// TIA Portal V15.1 export
// export: Created 2024-05-17T05:38:21.716242Z, ExportSetting WithDefaults, DisplayName Totally Integrated Automation Portal, DisplayVersion V15.1 Update 5, DisplayName TIA Portal Openness, DisplayVersion V15.1 Update 5, DisplayName SINAMICS Startdrive Advanced, DisplayVersion V15.1, DisplayName G130, G150, S120, S150, SINAMICS MV, S210, DisplayVersion V15.1, DisplayName G110M, G120, G120C, G120D, G120P, DisplayVersion V15.1, DisplayName STEP 7 Professional, DisplayVersion V15.1 Update 5, DisplayName STEP 7 Safety, DisplayVersion V15.1, DisplayName WinCC Professional, DisplayVersion V15.1 Update 5, DisplayName SIMATIC Visualization Architect, DisplayVersion V15.1
DATA_BLOCK "_209230ZS01ModeSummary"   // DB1901
{ S7_Optimized_Access := 'TRUE' }
AUTHOR : CSTAAL
VERSION : 0.1
// stored: AutoNumber false, DBAccessibleFromOPCUA true, InstanceOfName LModeSummary, InstanceOfType FB
"LModeSummary"
   // VAR_OUTPUT
   //    O_SumAutoMode { ExternalAccessible := 'False'; ExternalVisible := 'False'; ExternalWritable := 'False'} : Bool;
   //    O_SumAutoModeSel { ExternalAccessible := 'False'; ExternalVisible := 'False'; ExternalWritable := 'False'} : Bool;
   //    O_SumStepMode { ExternalAccessible := 'False'; ExternalVisible := 'False'; ExternalWritable := 'False'} : Bool;
   //    O_SumStepModeSel { ExternalAccessible := 'False'; ExternalVisible := 'False'; ExternalWritable := 'False'} : Bool;
   //    O_SumHomeRunMode { ExternalAccessible := 'False'; ExternalVisible := 'False'; ExternalWritable := 'False'} : Bool;
   //    O_SumHomeRunModeSel { ExternalAccessible := 'False'; ExternalVisible := 'False'; ExternalWritable := 'False'} : Bool;
   //    O_SumManualMode { ExternalAccessible := 'False'; ExternalVisible := 'False'; ExternalWritable := 'False'} : Bool;
   //    O_SumManualModeSel { ExternalAccessible := 'False'; ExternalVisible := 'False'; ExternalWritable := 'False'} : Bool;
   //    O_SumAnyProdModeActive { ExternalAccessible := 'False'; ExternalVisible := 'False'; ExternalWritable := 'False'} : Bool;
   //    O_SumAnyProdModeSel { ExternalAccessible := 'False'; ExternalVisible := 'False'; ExternalWritable := 'False'} : Bool;
   //    O_SumMode { ExternalAccessible := 'False'; ExternalVisible := 'False'; ExternalWritable := 'False'} : "Modes";
   // END_VAR
   // VAR_IN_OUT
   //    IO_ModesZM1 : "Modes";
   //    IO_ModesZM2 : "Modes";
   //    IO_ModesZM3 : "Modes";
   //    IO_ModesZM4 : "Modes";
   //    IO_ModesZM5 : "Modes";
   // END_VAR
BEGIN
END_DATA_BLOCK
